SUBAPPLICATION Uebung_002a (* DigitalInput_I1/_I2 auf DigitalOutput_Q1 *)
  (* Standard: 61499-2; Description: Copyright (c) 2023 Meisterschulen am Ostbahnhof This program and the accompanying materials are made available under the terms of the Eclipse Public License 2.0 which is available at https://www.eclipse.org/legal/epl-2.0/ SPDX-License-Identifier: EPL-2.0 *)
  (* Version 1.0, 2023-10-23, Franz Höpfinger, Meisterschulen am Ostbahnhof *)
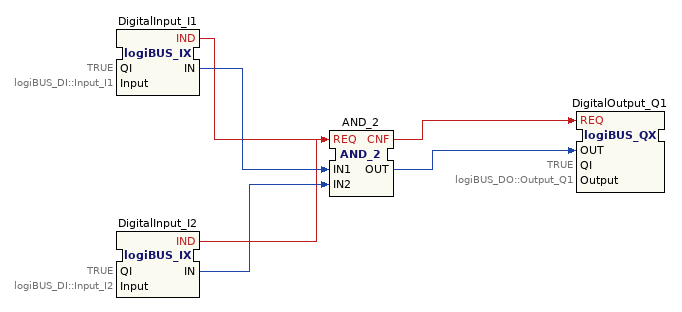
  FBS
    DigitalOutput_Q1 : logiBUS_QX(QI := TRUE, Output := logiBUS_DO::Output_Q1);
    DigitalInput_I1 : logiBUS_IX(QI := TRUE, Input := logiBUS_DI::Input_I1);
    DigitalInput_I2 : logiBUS_IX(QI := TRUE, Input := logiBUS_DI::Input_I2);
    AND_2 : AND_2;
  END_FBS
  EVENT_CONNECTIONS
    DigitalInput_I1.IND TO AND_2.REQ;
    DigitalInput_I2.IND TO AND_2.REQ;
    AND_2.CNF TO DigitalOutput_Q1.REQ;
  END_CONNECTIONS
  DATA_CONNECTIONS
    AND_2.OUT TO DigitalOutput_Q1.OUT;
    DigitalInput_I1.IN TO AND_2.IN1;
    DigitalInput_I2.IN TO AND_2.IN2;
  END_CONNECTIONS
END_SUBAPPLICATION
